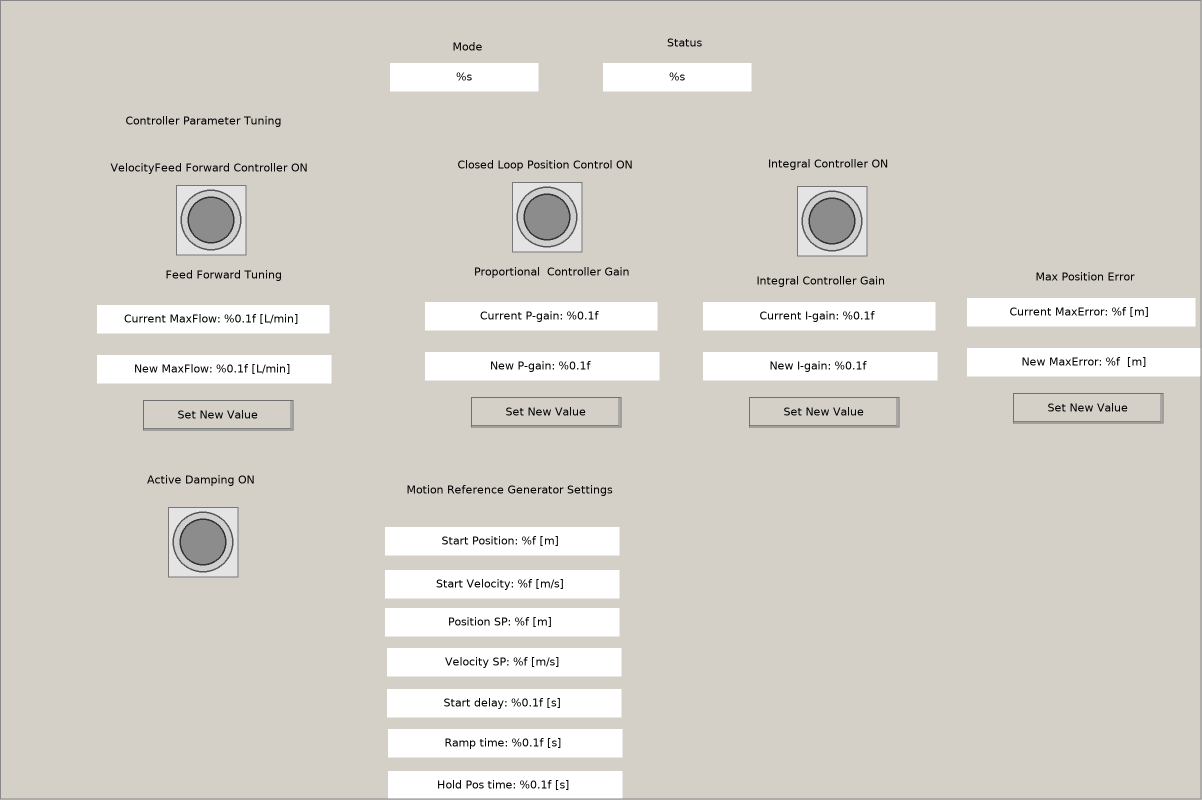
VISUALIZATION CommissioningHMI  // 1202x800
    Button (471,397 150x30), "Set New Value"
        tap G_Commissioning.bSetNewProportionalGain
    Textfield (424,301 234x30), "Current P-gain: %0.1f", text variable: G_Parameters.stParam.stClosedLoopControlSettings.fProportionalGain
    Textfield (424,351 236x30), "New P-gain: %0.1f", text variable: G_Commissioning.fNewProportionalGain
        OnMouseDown: write the text variable via Default
    Label (469,257 166x30), "Proportional Controller Gain"
    Button (749,397 150x30), "Set New Value"
        tap G_Commissioning.bSetNewIntegralGain
    Textfield (702,301 234x30), "Current I-gain: %0.1f", text variable: G_Parameters.stParam.stClosedLoopControlSettings.fIntegralGain
    Textfield (702,351 236x30), "New I-gain: %0.1f", text variable: G_Commissioning.fNewIntegralGain
        OnMouseDown: write the text variable via Default
    Label (746,266 150x30), "Integral Controller Gain"
    Label (94,106 219x30), "Controller Parameter Tuning"
    PushSwitch (797,186 70x70), variable: G_Commissioning.stAutomaticControlSettings.bEnableIntegralController, behaviour: TOGGLE, style: Switch-PushSwitch-Gray
    Label (745,149 166x30), "Integral Controller ON"
    Label (419,150 252x30), "Closed Loop Position Control ON"
    PushSwitch (512,182 70x70), variable: G_Commissioning.stAutomaticControlSettings.bEnableClosedLoopPositionControl, behaviour: TOGGLE, style: Switch-PushSwitch-Gray
    Label (83,153 252x30), "VelocityFeed Forward Controller ON"
    PushSwitch (176,185 70x70), variable: G_Commissioning.stAutomaticControlSettings.bEnableVelocityFeedForwardControl, behaviour: TOGGLE, style: Switch-PushSwitch-Gray
    PushSwitch (168,507 70x70), variable: G_Commissioning.stAutomaticControlSettings.bEnableActiveDamping, behaviour: TOGGLE, style: Switch-PushSwitch-Gray
    Label (75,465 252x30), "Active Damping ON"
    Button (143,400 150x30), "Set New Value"
        tap G_Commissioning.bSetNewMaxFlowCapacity
    Textfield (96,304 234x30), "Current MaxFlow: %0.1f [L/min]", text variable: G_Parameters.stParam.stOpenLoopControlSettings.fMaxFlowCapacity
    Textfield (96,354 236x30), "New MaxFlow: %0.1f [L/min]", text variable: G_Commissioning.fNewMaxFlowCapacity
        OnMouseDown: write the text variable via Default, min 0, max 40
    Label (141,260 166x30), "Feed Forward Tuning"
    Button (1013,393 150x30), "Set New Value"
        tap G_Commissioning.bSetNewMaxPositionError
    Textfield (966,297 230x30), "Current MaxError: %f [m]", text variable: G_Parameters.stParam.stClosedLoopControlSettings.fMaxPositionError
    Textfield (966,347 236x30), "New MaxError: %f [m]", text variable: G_Commissioning.fNewMaxPositionError
        OnMouseDown: write the text variable via Default
    Label (1010,262 150x30), "Max Position Error"
    Label (412,32 111x30), "Mode"
    Label (629,28 111x30), "Status"
    Textfield (389,62 150x30), "%s", text variable: G_Work.eMode
    Textfield (602,62 150x30), "%s", text variable: G_Work.eStatus
    Label (364,475 291x30), "Motion Reference Generator Settings"
    Textfield (384,526 236x30), "Start Position: %f [m]", text variable: G_Commissioning.stMotionReferenceGeneratorSettings.fStartPosition_m
        OnMouseDown: write the text variable via Default, min 0, max 0.5
    Textfield (384,569 236x30), "Start Velocity: %f [m/s]", text variable: G_Commissioning.stMotionReferenceGeneratorSettings.fStartVelocity_m
        OnMouseDown: write the text variable via Default, min 0, max 0.05
    Textfield (384,607 236x30), "Position SP: %f [m]", text variable: G_Commissioning.stMotionReferenceGeneratorSettings.fPositionSetpoint_ms
        OnMouseDown: write the text variable via Default, min 0, max 0.45
    Textfield (386,647 236x30), "Velocity SP: %f [m/s]", text variable: G_Commissioning.stMotionReferenceGeneratorSettings.fVelocitySetpoint_m
        OnMouseDown: write the text variable via Default, min 0, max 0.05
    Textfield (386,688 236x30), "Start delay: %0.1f [s]", text variable: G_Commissioning.stMotionReferenceGeneratorSettings.fTimeBeforeStarting_s
        OnMouseDown: write the text variable via Default, min 0, max 10
    Textfield (387,728 236x30), "Ramp time: %0.1f [s]", text variable: G_Commissioning.stMotionReferenceGeneratorSettings.fRampTime_s
        OnMouseDown: write the text variable via Default, min 0, max 10
    Textfield (387,770 236x30), "Hold Pos time: %0.1f [s]", text variable: G_Commissioning.stMotionReferenceGeneratorSettings.fHoldPositionTime_s
        OnMouseDown: write the text variable via Default, min 0, max 10
END_VISUALIZATION

(* stored: Version 1.1.0.1, ProductVersion 3.1.4024.10
   Visu CommissioningHMI: Id {bd8078e2-e5c4-4da6-a0a9-f1f5bbab114b} *)
